{attribute clr[Container(Layout.Stack)]}
{attribute clr[Group(Layout.GroupBox)]}
{attribute addProperty PreviousPort "Unknown"}
TYPE EtcSlaveTerminalBase_947E5A46 :
STRUCT
END_STRUCT
END_TYPE

(* stored: Version 1.2.0.0, ProductVersion 3.1.4024.9
   DUT EtcSlaveTerminalBase_947E5A46: Id {1caf7f9a-6561-4619-835e-dcd7aec91567} *)
